INTERFACE I_ListLogger

METHOD PUBLIC M_Add : BOOL
VAR_INPUT
	Object: 	I_Logger;
END_VAR
END_METHOD

METHOD PUBLIC M_Clear : BOOL
END_METHOD

METHOD PUBLIC M_Find : DINT
VAR_INPUT
	Object: 	I_Logger;
END_VAR
END_METHOD

METHOD PUBLIC M_Index : I_Logger
VAR_INPUT
	Index: 	DINT;
END_VAR
END_METHOD

METHOD PUBLIC M_Remove : BOOL
VAR_INPUT
	Object: 	I_Logger;
END_VAR
END_METHOD

{attribute 'OPC.UA.DA.Property' := '1'}
{attribute 'monitoring' := 'call'}
PROPERTY public P_Length : DINT
GET
END_GET
END_PROPERTY

END_INTERFACE

(* stored: Version 1.1.0.1
   Itf I_ListLogger: Id {3804175e-5c23-4e85-851d-b46040f3d4fc}
   Method M_Add: Id {bb6894bd-95db-4dfc-a37c-4551f8c81996}
   Method M_Clear: Id {42b944fe-c4e9-4d67-8d8d-2d21efb26ca5}
   Method M_Find: Id {27ece2d1-245f-4305-b083-0725d49d1055}
   Method M_Index: Id {374ba7bd-3bec-4072-b499-606ddd19a8d2}
   Method M_Remove: Id {82f6a8d9-07ac-4ed2-87eb-9f351254f787}
   Property P_Length: Id {51ce75fa-8eec-4323-94be-787fb7a7b131}
   Get Get: Id {94467135-43e8-4166-9086-021edefd1dcb} *)
